FUNCTION_BLOCK StringBuilderInfinite
VAR
	_Capacity : DINT;
	_Length : DINT;
	_Value : POINTER TO STRING := Allocate();
END_VAR
VAR CONSTANT
	InitialCapacity : DINT := 1024;
END_VAR

METHOD PRIVATE Allocate : POINTER TO STRING
VAR
	p : POINTER TO STRING;
END_VAR
_Capacity := InitialCapacity;
p := __NEW(BYTE, TO_UDINT(_Capacity + 1));
MEMSET(destAddr := p, fillByte := 0, n := TO_UDINT(_Capacity));
Allocate := p;
END_METHOD

METHOD Append : REFERENCE TO StringBuilderInfinite
VAR_INPUT
	value : T_MaxString;
END_VAR
VAR
	lengthToCopy : DINT;
END_VAR
lengthToCopy := LEN(value);

EnsureCapacity(_Length + lengthToCopy);

MEMCPY(
	destAddr := _Value + _Length,
	srcAddr := ADR(value),
	n := TO_UDINT(lengthToCopy)
);

_Length := _Length + lengthToCopy;

Append REF= THIS^;
END_METHOD

METHOD AppendByPointer : REFERENCE TO StringBuilderInfinite
VAR_INPUT
	value : POINTER TO STRING;
END_VAR
VAR
	lengthToCopy : DINT;
END_VAR
lengthToCopy := TO_DINT(LEN2(value));

EnsureCapacity(_Length + lengthToCopy);

MEMCPY(
	destAddr := _Value + TO_LWORD(_Length),
	srcAddr := value,
	n := TO_UDINT(lengthToCopy)
);

_Length := _Length + lengthToCopy;

AppendByPointer REF= THIS^;
END_METHOD

{attribute 'monitoring' := 'call'}
PROPERTY Capacity : DINT
GET
Capacity := _Capacity;
END_GET
END_PROPERTY

METHOD Clear : REFERENCE TO StringBuilderInfinite
MEMSET(
	destAddr := _Value,
	fillByte := 0,
	n := TO_UDINT(_Length)
);

_Length := 0;

Clear REF= THIS^;
END_METHOD

METHOD PRIVATE EnsureCapacity
VAR_INPUT
	needed : DINT;
END_VAR
IF (needed < _Capacity) THEN
	RETURN;
END_IF

IF (needed > _Capacity * 2) THEN
	_Capacity := needed;
ELSE
	_Capacity := NextPowerOf2(needed);
END_IF

Reallocate();
END_METHOD

METHOD FB_exit : BOOL
VAR_INPUT
	bInCopyCode : BOOL; // if TRUE, the exit method is called for exiting an instance that is copied afterwards (online change).
END_VAR
__DELETE(_Value);
END_METHOD

PROPERTY IsEmpty : BOOL
GET
IsEmpty := Length = 0;
END_GET
END_PROPERTY

{attribute 'monitoring' := 'call'}
PROPERTY Length : DINT
GET
Length := _Length;
END_GET
END_PROPERTY

METHOD PRIVATE NextPowerOf2 : DINT
VAR_INPUT
	number : DINT;
END_VAR
VAR
	n : UDINT;
END_VAR
n := TO_UDINT(number);
n := n - 1;
n := n OR SHR(n, 1);
n := n OR SHR(n, 2);
n := n OR SHR(n, 4);
n := n OR SHR(n, 8);
n := n OR SHR(n, 16);
n := n + 1;
NextPowerOf2 := TO_DINT(n);
END_METHOD

METHOD PRIVATE Reallocate
VAR_INPUT
END_VAR
VAR
	new : POINTER TO STRING;
END_VAR
new := __NEW(BYTE, TO_UDINT(_Capacity + 1));
MEMSET(destAddr := new, fillByte := 0, n := TO_UDINT(_Capacity));
MEMCPY(new, _Value, TO_UDINT(_Length));
__DELETE(_Value);
_Value := new;
END_METHOD

{attribute 'monitoring' := 'call'}
PROPERTY Value : POINTER TO STRING(1000)
GET
Value := _Value;
END_GET
END_PROPERTY

END_FUNCTION_BLOCK

(* stored: Version 1.1.0.1
   POU StringBuilderInfinite: Id {494d6245-e98b-407b-8559-a62542a9481d}, SpecialFunc None
   Method Allocate: Id {72f372ee-36a0-4599-bcb3-9e89a2e7d55f}
   Method Append: Id {3f970321-6f9c-4ccc-a49e-0bee078cd44e}
   Method AppendByPointer: Id {e006be62-c9ae-42f9-8fa8-db175748148b}
   Property Capacity: Id {c6065eee-19df-405d-9144-9537f9fd3d36}
   Get Get: Id {82a87c1d-357d-4e74-9854-e7f5ff606f38}
   Method Clear: Id {1c371b6f-9ba8-42e2-be37-4fe7f206e4c7}
   Method EnsureCapacity: Id {b4d61f91-eb48-4a47-a69f-a556c9b5aa5e}
   Method FB_exit: Id {089b2b60-5868-4471-8e05-d2e1026c18e5}
   Property IsEmpty: Id {d36d74ea-bcac-4b88-9ef3-3fe5ee91e2e3}
   Get Get: Id {5c965a97-5668-4cf4-8e11-ba178f6b9362}
   Property Length: Id {2bbbae11-4f2c-44c2-b6cc-708c2ab7daf4}
   Get Get: Id {ac7f521b-1ab7-44a1-b536-c1b960a89b90}
   Method NextPowerOf2: Id {3b448972-0092-4aa9-ae1a-997eaf88648a}
   Method Reallocate: Id {8f039273-b116-47dd-bf35-078db7701848}
   Property Value: Id {cfdb86ac-3c93-4424-b346-f83099aa6553}
   Get Get: Id {8a91e9a7-9267-487a-87eb-3359d3a82716} *)
